INTERFACE ITF_TopElement2_HMI_Connector EXTENDS ITF_BaseTopElement_HMI_Connector,
	ITF_TopElement2_HMI_Connector_View, ITF_TopElement2_HMI_Connector_Command

END_INTERFACE

(* stored: Version 1.1.0.1
   Itf ITF_TopElement2_HMI_Connector: Id {58efa8a6-3ccd-06c9-128c-7b8c049cd710} *)
